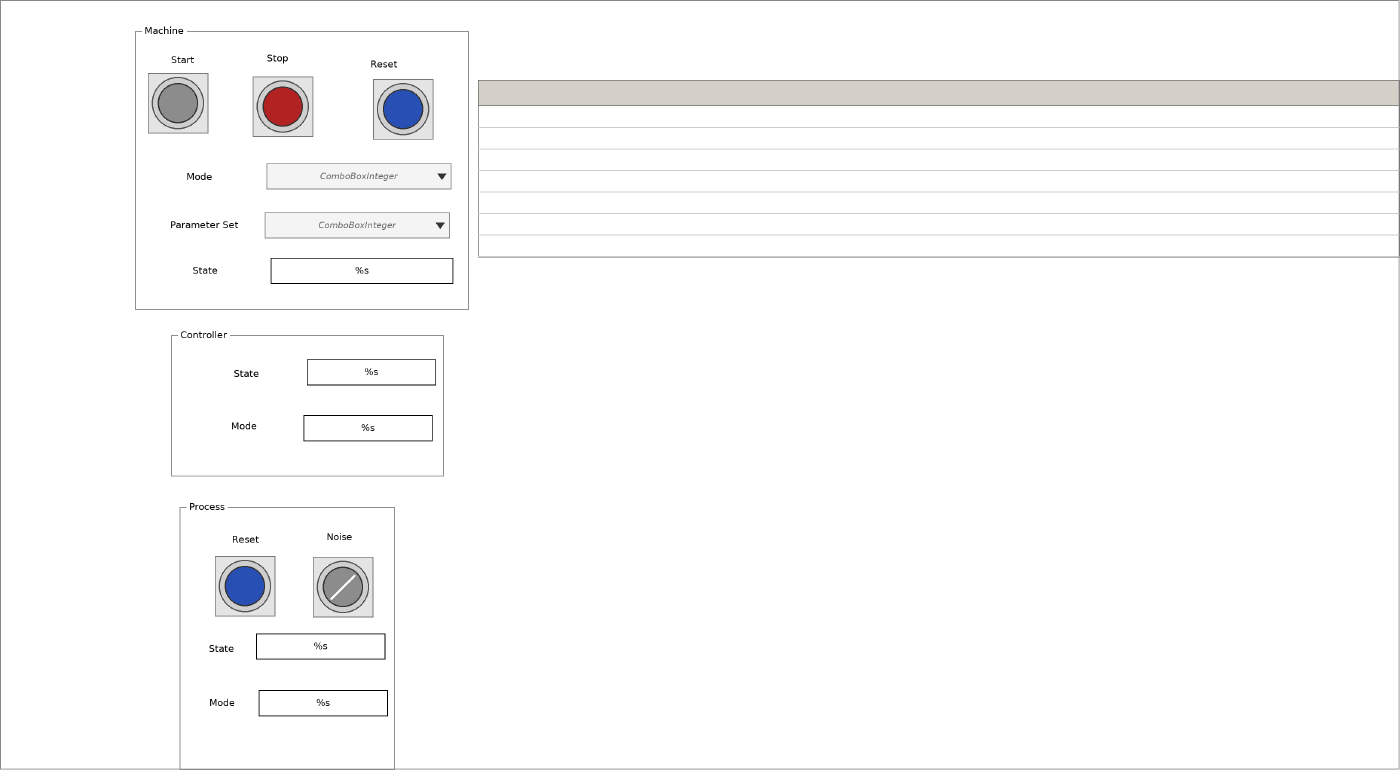
VISUALIZATION Visualization  // 1629x896
    GroupBox (199,382 317x172), "Controller"
        Rectangle (158,36 150x30), "%s", text variable: MAIN.sControllerState
        Label (13,38 150x30), "State"
        Label (10,99 150x30), "Mode"
        Rectangle (154,101 150x30), "%s", text variable: MAIN.sControllerMode
    GroupBox (209,582 250x314), "Process"
        PushSwitch (41,65 70x70), variable: MAIN.ResetProcess, behaviour: TAP, style: Switch-PushSwitch-Blue
        RotarySwitch (155,66 70x70), variable: MAIN.fbProcess.bNoise, behaviour: TOGGLE, style: Switch-RotarySwitch-Gray
        Label (2,31 150x30), "Reset"
        Rectangle (89,155 150x30), "%s", text variable: MAIN.sProcessStateHMI
        Rectangle (92,221 150x30), "%s", text variable: MAIN.sProcessModeHMI
        Label (145,28 82x30), "Noise"
        Label (13,158 72x30), "State"
        Label (9,221 81x30), "Mode"
    GroupBox (157,28 388x332), "Machine"
        PushSwitch (15,57 70x70), variable: MAIN.Start, behaviour: TAP, style: Switch-PushSwitch-Gray
        PushSwitch (137,61 70x70), variable: MAIN.Stop, behaviour: TAP, style: Switch-PushSwitch-Red
        Label (91,25 150x30), "Stop"
        PushSwitch (277,64 70x70), variable: MAIN.Reset, behaviour: TAP, style: Switch-PushSwitch-Blue
        Label (215,32 150x30), "Reset"
        ComboBoxInteger (153,162 215x30), variable: MAIN.Mode, text list: 'TL_Mode'
        Label (0,163 150x30), "Mode"
        ComboBoxInteger (151,219 215x30), variable: MAIN.SelectedParameterSet, text list: 'TL_SelectedParameterSet'
        Rectangle (158,272 212x30), "%s", text variable: MAIN.sState
        Label (7,272 150x30), "State"
        Label (10,27 91x30), "Start"
        Label (6,219 150x30), "Parameter Set"
    Table (556,93 1073x206), data array: MAIN.arControllerParams
        p3854506369: MAIN.arControllerParams[INDEX].KpHeat
        p1892666644: MAIN.arControllerParams[INDEX].TnHeat
        p338671338: MAIN.arControllerParams[INDEX].TvHeat
        p2170511999: MAIN.arControllerParams[INDEX].TdHeat
        p3723444502: MAIN.arControllerParams[INDEX].KpCool
        p1218418051: MAIN.arControllerParams[INDEX].TnCool
        p746581629: MAIN.arControllerParams[INDEX].TvCool
        p3104783080: MAIN.arControllerParams[INDEX].TdCool
END_VISUALIZATION

(* stored: Version 1.1.0.1, ProductVersion 3.1.4024.12
   Visu Visualization: Id {86287df9-c8d9-437b-bd36-8168328efe30} *)
